(* Schneider Machine Expert - Basic project cb(1), file version 2.6.0.0 *)
(* ProjectInformations: Name=New project *)

HARDWARE
  Cpu 0: TM221CE40R
  EthernetConfiguration: NetworkName=M221, IpAllocationMode=FixedAddress, IpAddress=192.168.0.2, SubnetMask=255.255.255.0
  SerialLineConfiguration: Baud=Baud19200, Parity=ParityEven, DataBits=DataBits8, StopBits=StopBits1, PhysicalMedium=PhysicalMediumRs485, TransmissionMode=TransmissionModeModbusRtu, SlaveId=1, Addressing=SlaveAddressing
  MastTask: UsePeriodScanMode=false, PeriodScan=100
  FastTask: Period=255
  CpuBehavior: StartingMode=StartAsPreviousState, AutoSaveRamOnEeprom=true, WatchdogPeriod=250

SYMBOLS  (address, symbol, comment, settings)
  %M0         "START"
  %M1         "MOVE_TRF"
  %M2         "GRIPPER_C_CLOSE"
  %M3         "MOVE_BACK_TRF"
  %M4         "GRIPPER_ROTATE_CLOSE"
  %M5         "STATUS CB ON"
  %M6         "RELEASE_C_GRIPPER"
  %M7         "POLARITY_ RESULT"
  %M8         "POLARITY_CHECK"
  %M9         "ROTATE_0"
  %M10        "REVERSE_ROTATION"
  %M11        "RESET"
  %M12        "MANUAL"
  %M13        "CB_LF"
  %M14        "CB_RT"
  %M15        "DELAY_CUT_LEFT"
  %M16        "Cut Left"
  %M17        "Cut Right"
  %M19        "Grimp Comp"
  %M20        "R_Grip"
  %M21        "Slide"
  %M22        "LF_CB"
  %M23        "M_Q1"
  %M24        "M_Q2"
  %M25        "M_Q3"
  %M26      MANUAL_GRIP_CLOSE  "M_Q4"
  %M27      SLIDER  "M_Q5"
  %M28        "M_Q6"
  %M29        "Manual Bowl"
  %M30        "EMG_Memory"
  %M31        "Start_Memory"
  %M47        "M_EMG"
  %M49        "POLARITY CHECKED"
  %M50        "NEGATIVE"
  %M51        "POSITIVE"
  %M52        "FIRST RUN"
  %M53        "DONE CUTTING"
  %M54        "NEGATIVE READY"
  %M55        "TRIGGER"
  %M56        "COUNTER OUTPUT"
  %M100       "START GUI"
  %M102       "M_START"
  %MW0        "Count Output"
  %TM0        [Preset=50, Base=TenMilliSeconds]
  %TM1        [Preset=10, Base=TenMilliSeconds]
  %TM2        "Left Cut"  [Preset=10, Base=TenMilliSeconds]
  %I0.0       "EMG"
  %I0.1       "BTN START"
  %I0.2       "LF_CB_FWD"
  %I0.3       "LF_CB_BWD"
  %I0.4       "RT_CB_FWD"
  %I0.5       "RT_CB_BWD"
  %I0.6       "R_CW"
  %I0.7       "R_CCW"
  %I0.8       "GRIP_R_OPEN"
  %I0.9       "GRIP_R_CLOSE"
  %I0.10      "GRIP_C_OPEN"
  %I0.11      "GRIP_C_CLOSE"
  %I0.12      "C_TRF_FWD"
  %I0.13      "TRF_C_BWD"
  %I0.14      "PART_DETECTION"
  %I0.15      "GRIP_C_OPEN"
  %I0.16      "GRIP_C_OPEN"
  %I0.19      "BUTTON POLARITY"
  %Q0.0       "LF_CB"
  %Q0.1       "RT_CB"
  %Q0.2       "R_P"
  %Q0.3       "GRIP_COMP"
  %Q0.4       "GRIP_ROTATE"
  %Q0.5       "TRF_C"
  %Q0.6       "BOWL_FEEDER"

POU New POU
  (* SectionNumber=1 *)

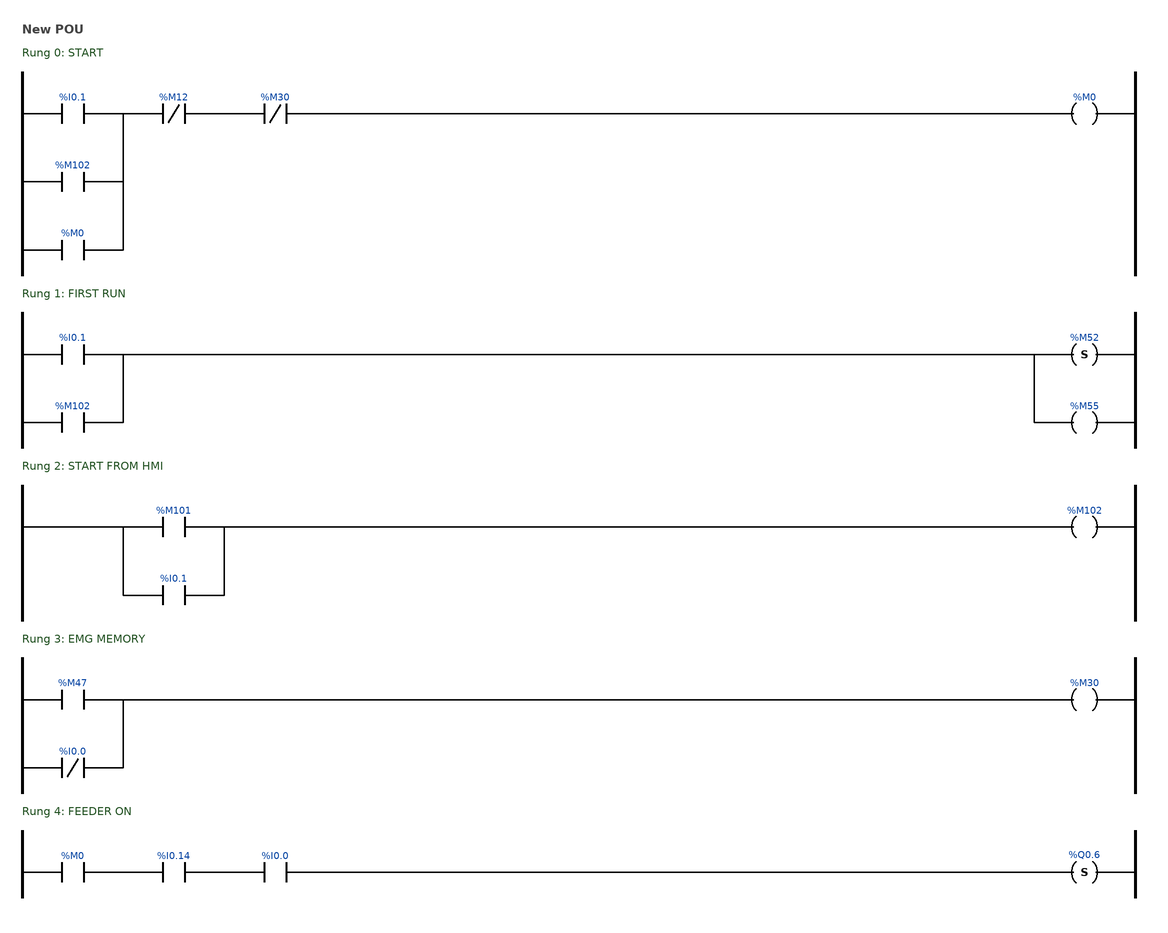

// Rung 0: START
  LD %I0.1
  OR %M102
  OR %M0
  ANDN %M12
  ANDN %M30
  ST %M0
  // as ST:
  //   %M0 := (%I0.1 OR %M102 OR %M0) AND NOT %M12 AND NOT %M30;

// Rung 1: FIRST RUN
  LD %I0.1
  OR %M102
  S %M52
  ST %M55
  // as ST:
  //   IF %I0.1 OR %M102 THEN %M52 := TRUE; END_IF;
  //   %M55 := %I0.1 OR %M102;

// Rung 2: START FROM HMI
  LD 1
  AND( %M101
  OR %I0.1
  )
  ST %M102
  // as ST:
  //   %M102 := %M101 OR %I0.1;

// Rung 3: EMG MEMORY
  LD %M47
  ORN %I0.0
  ST %M30
  // as ST:
  //   %M30 := %M47 OR NOT %I0.0;

// Rung 4: FEEDER ON
  LD %M0
  AND %I0.14
  AND %I0.0
  S %Q0.6
  // as ST:
  //   IF %M0 AND %I0.14 AND %I0.0 THEN %Q0.6 := TRUE; END_IF;

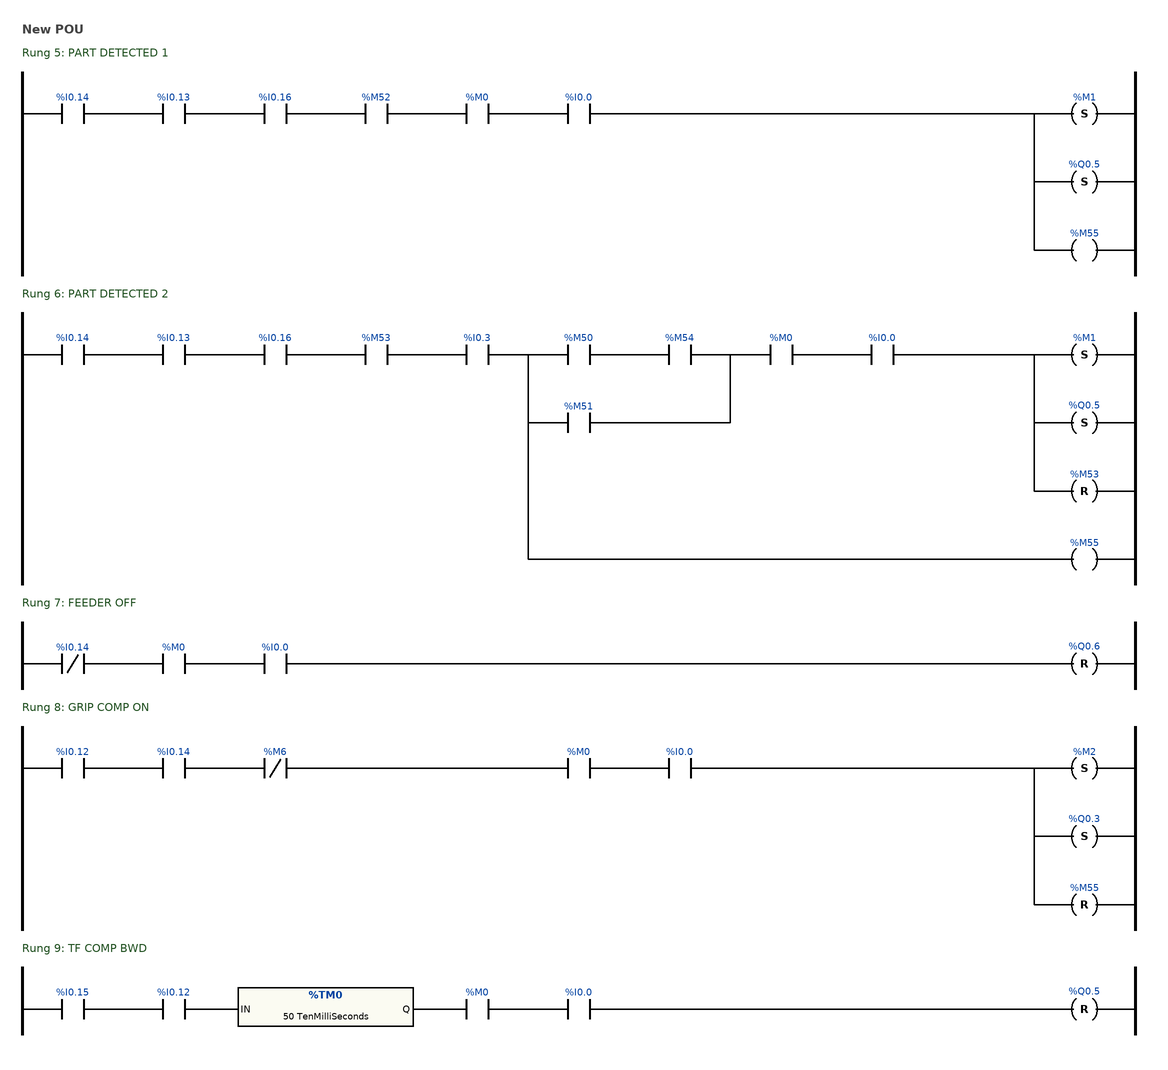

// Rung 5: PART DETECTED 1
  LD %I0.14
  AND %I0.13
  AND %I0.16
  AND %M52
  AND %M0
  AND %I0.0
  S %M1
  S %Q0.5
  ST %M55
  // as ST:
  //   IF %I0.14 AND %I0.13 AND %I0.16 AND %M52 AND %M0 AND %I0.0 THEN %M1 := TRUE; END_IF;
  //   IF %I0.14 AND %I0.13 AND %I0.16 AND %M52 AND %M0 AND %I0.0 THEN %Q0.5 := TRUE; END_IF;
  //   %M55 := %I0.14 AND %I0.13 AND %I0.16 AND %M52 AND %M0 AND %I0.0;

// Rung 6: PART DETECTED 2
  LD %I0.14
  AND %I0.13
  AND %I0.16
  AND %M53
  AND %I0.3
  MPS
  AND( %M50
  AND %M54
  OR %M51
  )
  AND %M0
  AND %I0.0
  S %M1
  S %Q0.5
  R %M53
  MPP
  ST %M55
  // as ST:
  //   IF %I0.14 AND %I0.13 AND %I0.16 AND %M53 AND %I0.3 AND (%M50 AND %M54 OR %M51) AND %M0 AND %I0.0 THEN %M1 := TRUE; END_IF;
  //   IF %I0.14 AND %I0.13 AND %I0.16 AND %M53 AND %I0.3 AND (%M50 AND %M54 OR %M51) AND %M0 AND %I0.0 THEN %Q0.5 := TRUE; END_IF;
  //   _t1 := %I0.14 AND %I0.13 AND %I0.16 AND %M53 AND %I0.3;
  //   IF %I0.14 AND %I0.13 AND %I0.16 AND %M53 AND %I0.3 AND (%M50 AND %M54 OR %M51) AND %M0 AND %I0.0 THEN %M53 := FALSE; END_IF;
  //   %M55 := _t1;

// Rung 7: FEEDER OFF
  LDN %I0.14
  AND %M0
  AND %I0.0
  R %Q0.6
  // as ST:
  //   IF NOT %I0.14 AND %M0 AND %I0.0 THEN %Q0.6 := FALSE; END_IF;

// Rung 8: GRIP COMP ON
  LD %I0.12
  AND %I0.14
  ANDN %M6
  AND %M0
  AND %I0.0
  S %M2
  S %Q0.3
  R %M55
  // as ST:
  //   IF %I0.12 AND %I0.14 AND NOT %M6 AND %M0 AND %I0.0 THEN %M2 := TRUE; END_IF;
  //   IF %I0.12 AND %I0.14 AND NOT %M6 AND %M0 AND %I0.0 THEN %Q0.3 := TRUE; END_IF;
  //   IF %I0.12 AND %I0.14 AND NOT %M6 AND %M0 AND %I0.0 THEN %M55 := FALSE; END_IF;

// Rung 9: TF COMP BWD
  BLK %TM0
  LD %I0.15
  AND %I0.12
  IN
  OUT_BLK
  LD Q
  AND %M0
  AND %I0.0
  R %Q0.5
  END_BLK
  // as ST:
  //   %TM0(IN := %I0.15 AND %I0.12);
  //   IF %TM0.Q AND %M0 AND %I0.0 THEN %Q0.5 := FALSE; END_IF;

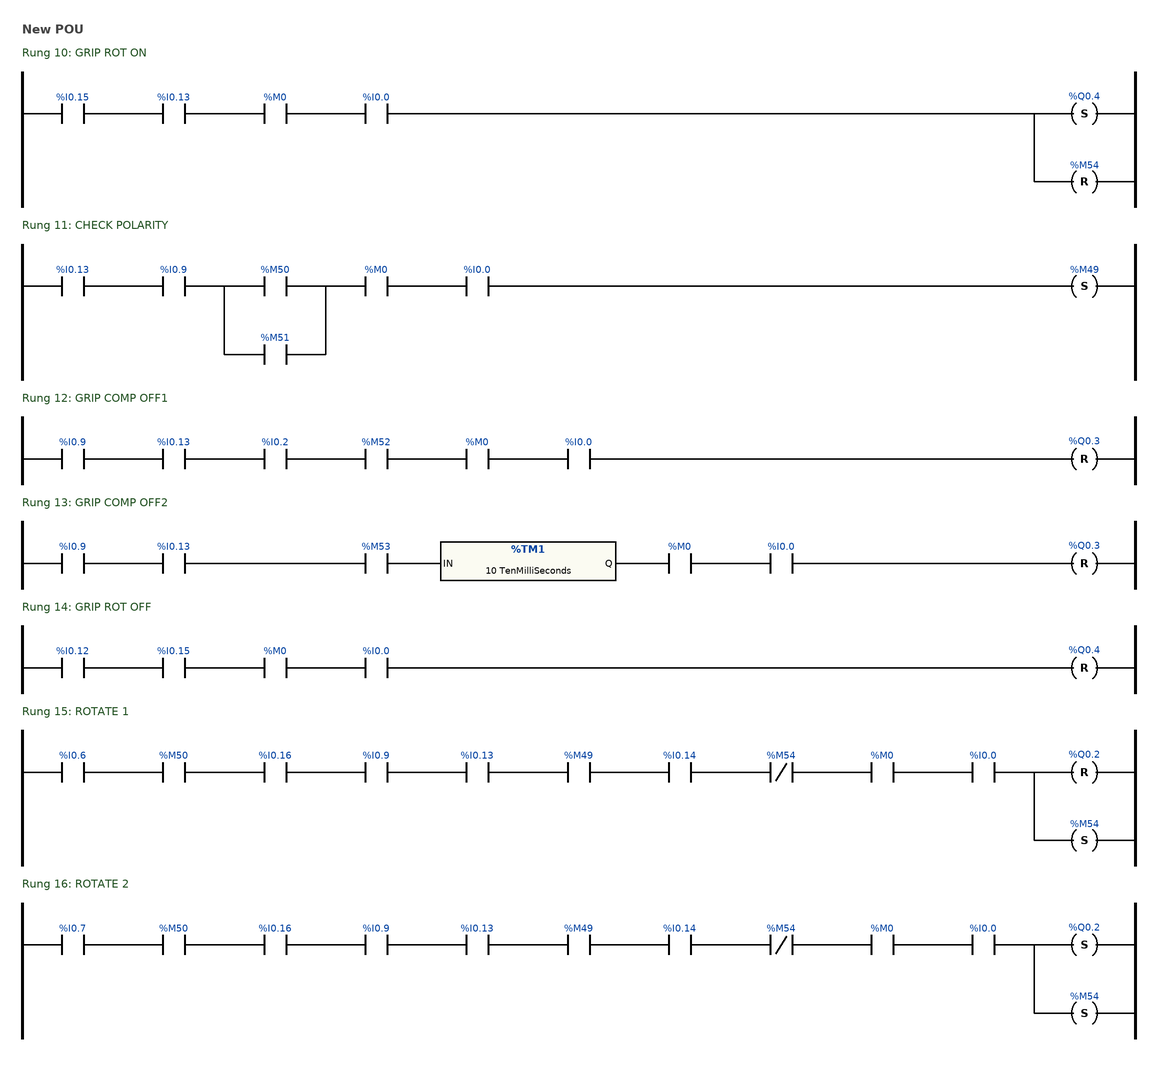

// Rung 10: GRIP ROT ON
  LD %I0.15
  AND %I0.13
  AND %M0
  AND %I0.0
  S %Q0.4
  R %M54
  // as ST:
  //   IF %I0.15 AND %I0.13 AND %M0 AND %I0.0 THEN %Q0.4 := TRUE; END_IF;
  //   IF %I0.15 AND %I0.13 AND %M0 AND %I0.0 THEN %M54 := FALSE; END_IF;

// Rung 11: CHECK POLARITY
  LD %I0.13
  AND %I0.9
  AND( %M50
  OR %M51
  )
  AND %M0
  AND %I0.0
  S %M49
  // as ST:
  //   IF %I0.13 AND %I0.9 AND (%M50 OR %M51) AND %M0 AND %I0.0 THEN %M49 := TRUE; END_IF;

// Rung 12: GRIP COMP OFF1
  LD %I0.9
  AND %I0.13
  AND %I0.2
  AND %M52
  AND %M0
  AND %I0.0
  R %Q0.3
  // as ST:
  //   IF %I0.9 AND %I0.13 AND %I0.2 AND %M52 AND %M0 AND %I0.0 THEN %Q0.3 := FALSE; END_IF;

// Rung 13: GRIP COMP OFF2
  BLK %TM1
  LD %I0.9
  AND %I0.13
  AND %M53
  IN
  OUT_BLK
  LD Q
  AND %M0
  AND %I0.0
  R %Q0.3
  END_BLK
  // as ST:
  //   %TM1(IN := %I0.9 AND %I0.13 AND %M53);
  //   IF %TM1.Q AND %M0 AND %I0.0 THEN %Q0.3 := FALSE; END_IF;

// Rung 14: GRIP ROT OFF
  LD %I0.12
  AND %I0.15
  AND %M0
  AND %I0.0
  R %Q0.4
  // as ST:
  //   IF %I0.12 AND %I0.15 AND %M0 AND %I0.0 THEN %Q0.4 := FALSE; END_IF;

// Rung 15: ROTATE 1
  LD %I0.6
  AND %M50
  AND %I0.16
  AND %I0.9
  AND %I0.13
  AND %M49
  AND %I0.14
  ANDN %M54
  AND %M0
  AND %I0.0
  R %Q0.2
  S %M54
  // as ST:
  //   IF %I0.6 AND %M50 AND %I0.16 AND %I0.9 AND %I0.13 AND %M49 AND %I0.14 AND NOT %M54 AND %M0 AND %I0.0 THEN %Q0.2 := FALSE; END_IF;
  //   IF %I0.6 AND %M50 AND %I0.16 AND %I0.9 AND %I0.13 AND %M49 AND %I0.14 AND NOT %M54 AND %M0 AND %I0.0 THEN %M54 := TRUE; END_IF;

// Rung 16: ROTATE 2
  LD %I0.7
  AND %M50
  AND %I0.16
  AND %I0.9
  AND %I0.13
  AND %M49
  AND %I0.14
  ANDN %M54
  AND %M0
  AND %I0.0
  S %Q0.2
  S %M54
  // as ST:
  //   IF %I0.7 AND %M50 AND %I0.16 AND %I0.9 AND %I0.13 AND %M49 AND %I0.14 AND NOT %M54 AND %M0 AND %I0.0 THEN %Q0.2 := TRUE; END_IF;
  //   IF %I0.7 AND %M50 AND %I0.16 AND %I0.9 AND %I0.13 AND %M49 AND %I0.14 AND NOT %M54 AND %M0 AND %I0.0 THEN %M54 := TRUE; END_IF;

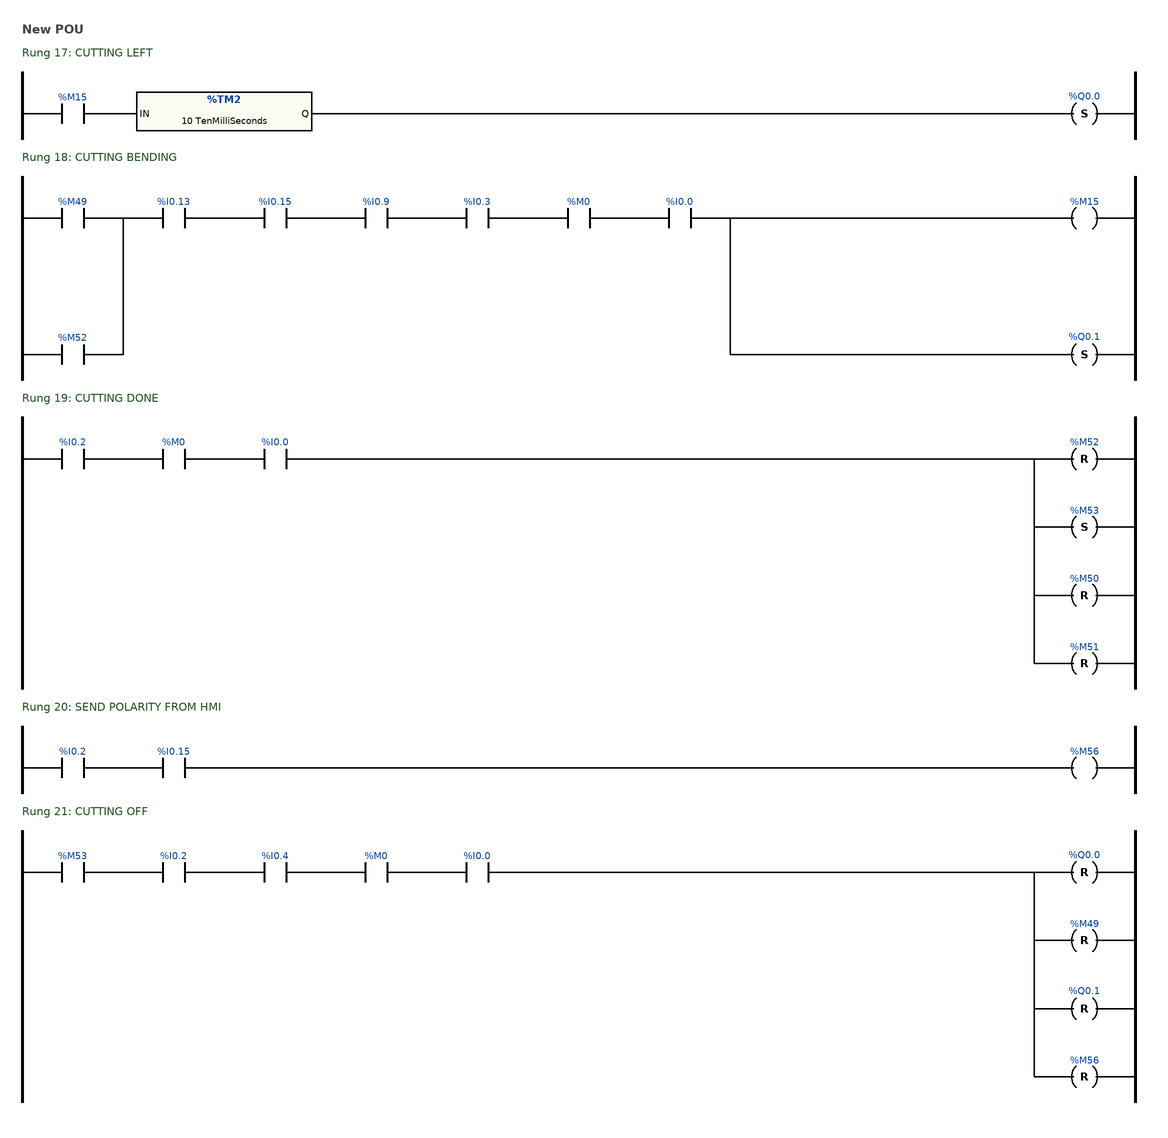

// Rung 17: CUTTING LEFT
  BLK %TM2
  LD %M15
  IN
  OUT_BLK
  LD Q
  S %Q0.0
  END_BLK
  // as ST:
  //   %TM2(IN := %M15);
  //   IF %TM2.Q THEN %Q0.0 := TRUE; END_IF;

// Rung 18: CUTTING BENDING
  LD %M49
  OR %M52
  AND %I0.13
  AND %I0.15
  AND %I0.9
  AND %I0.3
  AND %M0
  AND %I0.0
  ST %M15
  S %Q0.1
  // as ST:
  //   %M15 := (%M49 OR %M52) AND %I0.13 AND %I0.15 AND %I0.9 AND %I0.3 AND %M0 AND %I0.0;
  //   IF (%M49 OR %M52) AND %I0.13 AND %I0.15 AND %I0.9 AND %I0.3 AND %M0 AND %I0.0 THEN %Q0.1 := TRUE; END_IF;

// Rung 19: CUTTING DONE
  LD %I0.2
  AND %M0
  AND %I0.0
  R %M52
  S %M53
  R %M50
  R %M51
  // as ST:
  //   IF %I0.2 AND %M0 AND %I0.0 THEN %M52 := FALSE; END_IF;
  //   IF %I0.2 AND %M0 AND %I0.0 THEN %M53 := TRUE; END_IF;
  //   IF %I0.2 AND %M0 AND %I0.0 THEN %M50 := FALSE; END_IF;
  //   IF %I0.2 AND %M0 AND %I0.0 THEN %M51 := FALSE; END_IF;

// Rung 20: SEND POLARITY FROM HMI
  LD %I0.2
  AND %I0.15
  ST %M56
  // as ST:
  //   %M56 := %I0.2 AND %I0.15;

// Rung 21: CUTTING OFF
  LD %M53
  AND %I0.2
  AND %I0.4
  AND %M0
  AND %I0.0
  R %Q0.0
  R %M49
  R %Q0.1
  R %M56
  // as ST:
  //   IF %M53 AND %I0.2 AND %I0.4 AND %M0 AND %I0.0 THEN %Q0.0 := FALSE; END_IF;
  //   IF %M53 AND %I0.2 AND %I0.4 AND %M0 AND %I0.0 THEN %M49 := FALSE; END_IF;
  //   IF %M53 AND %I0.2 AND %I0.4 AND %M0 AND %I0.0 THEN %Q0.1 := FALSE; END_IF;
  //   IF %M53 AND %I0.2 AND %I0.4 AND %M0 AND %I0.0 THEN %M56 := FALSE; END_IF;

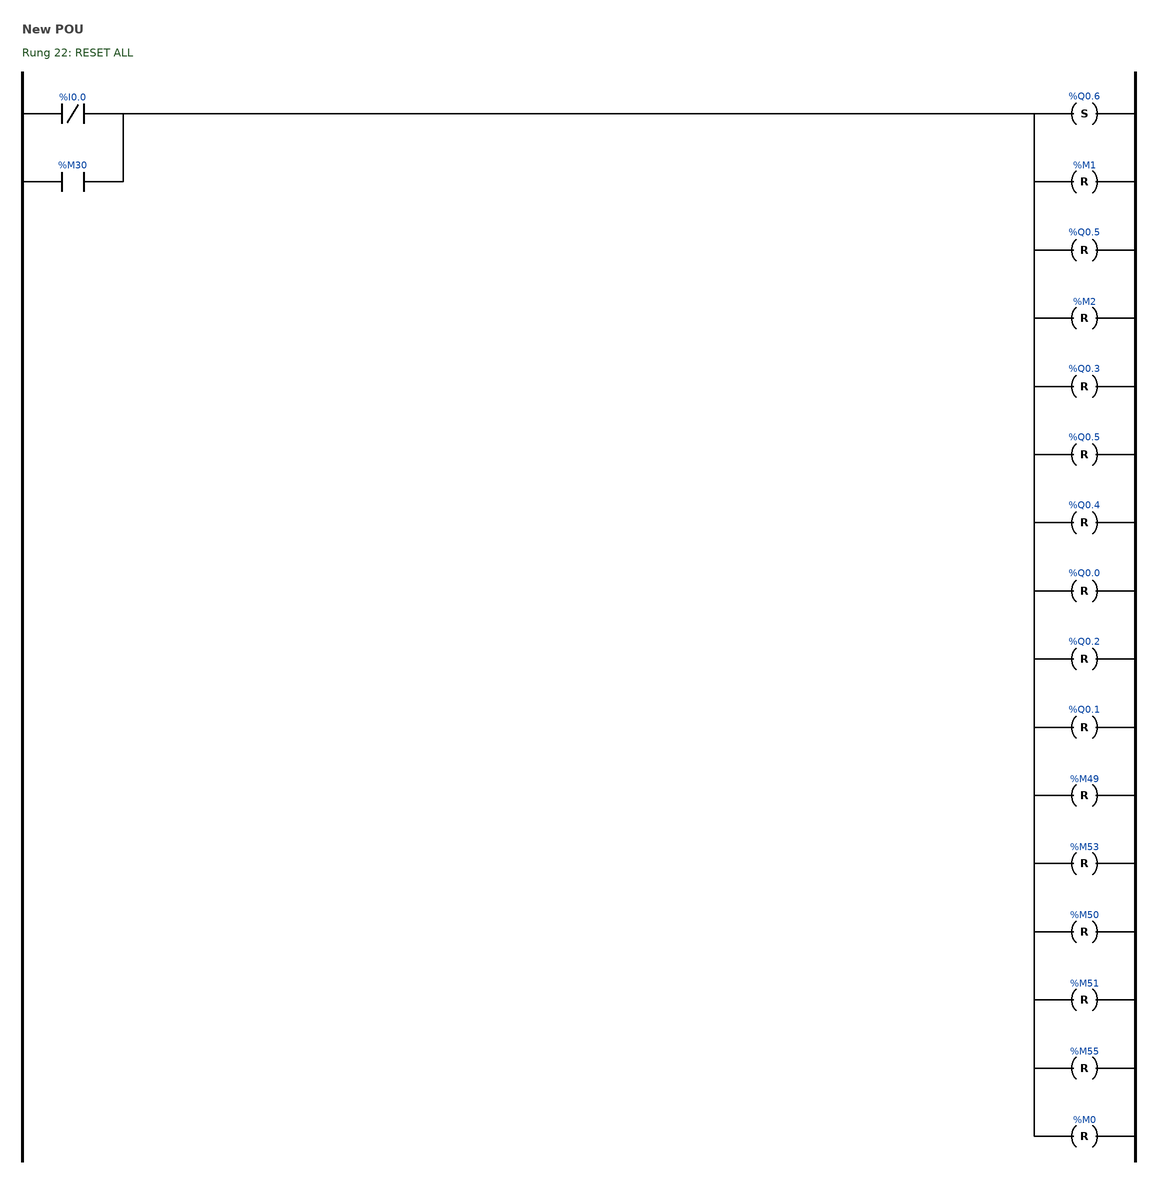

// Rung 22: RESET ALL
  LDN %I0.0
  OR %M30
  S %Q0.6
  R %M1
  R %Q0.5
  R %M2
  R %Q0.3
  R %Q0.5
  R %Q0.4
  R %Q0.0
  R %Q0.2
  R %Q0.1
  R %M49
  R %M53
  R %M50
  R %M51
  R %M55
  R %M0
  // as ST:
  //   IF NOT %I0.0 OR %M30 THEN %Q0.6 := TRUE; END_IF;
  //   IF NOT %I0.0 OR %M30 THEN %M1 := FALSE; END_IF;
  //   IF NOT %I0.0 OR %M30 THEN %Q0.5 := FALSE; END_IF;
  //   IF NOT %I0.0 OR %M30 THEN %M2 := FALSE; END_IF;
  //   IF NOT %I0.0 OR %M30 THEN %Q0.3 := FALSE; END_IF;
  //   IF NOT %I0.0 OR %M30 THEN %Q0.5 := FALSE; END_IF;
  //   IF NOT %I0.0 OR %M30 THEN %Q0.4 := FALSE; END_IF;
  //   IF NOT %I0.0 OR %M30 THEN %Q0.0 := FALSE; END_IF;
  //   IF NOT %I0.0 OR %M30 THEN %Q0.2 := FALSE; END_IF;
  //   IF NOT %I0.0 OR %M30 THEN %Q0.1 := FALSE; END_IF;
  //   IF NOT %I0.0 OR %M30 THEN %M49 := FALSE; END_IF;
  //   IF NOT %I0.0 OR %M30 THEN %M53 := FALSE; END_IF;
  //   IF NOT %I0.0 OR %M30 THEN %M50 := FALSE; END_IF;
  //   IF NOT %I0.0 OR %M30 THEN %M51 := FALSE; END_IF;
  //   IF NOT %I0.0 OR %M30 THEN %M55 := FALSE; END_IF;
  //   IF NOT %I0.0 OR %M30 THEN %M0 := FALSE; END_IF;

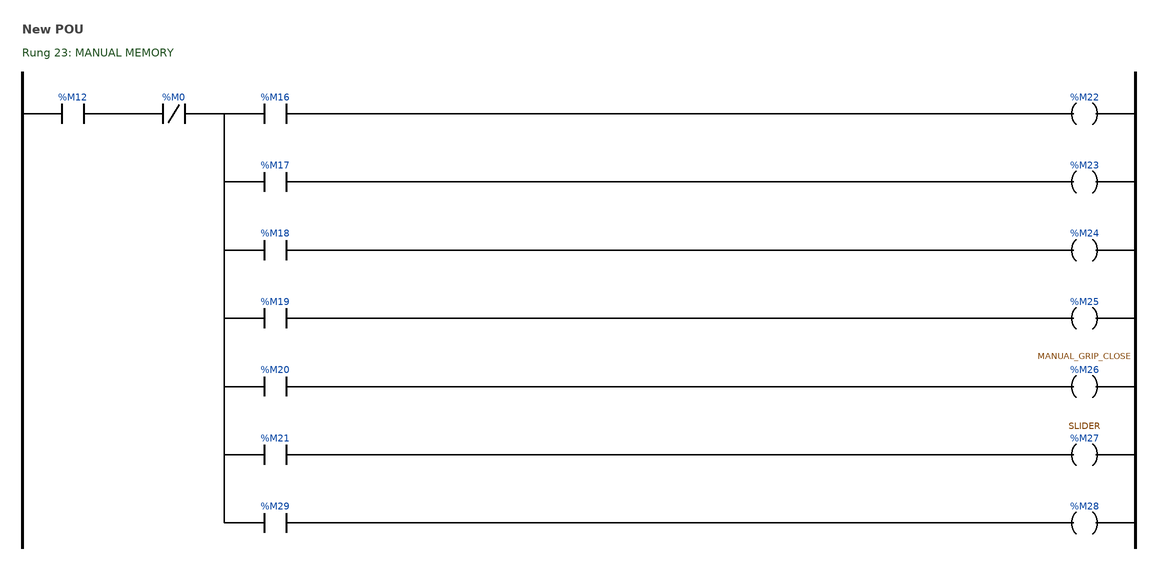

// Rung 23: MANUAL MEMORY
  LD %M12
  ANDN %M0
  MPS
  AND %M16
  ST %M22
  MRD
  AND %M17
  ST %M23
  MRD
  AND %M18
  ST %M24
  MRD
  AND %M19
  ST %M25
  MRD
  AND %M20
  ST %M26                 (* MANUAL_GRIP_CLOSE *)
  MRD
  AND %M21
  ST %M27                 (* SLIDER *)
  MPP
  AND %M29
  ST %M28
  // as ST:
  //   %M22 := %M12 AND NOT %M0 AND %M16;
  //   %M23 := %M12 AND NOT %M0 AND %M17;
  //   %M24 := %M12 AND NOT %M0 AND %M18;
  //   %M25 := %M12 AND NOT %M0 AND %M19;
  //   MANUAL_GRIP_CLOSE := %M12 AND NOT %M0 AND %M20;
  //   SLIDER := %M12 AND NOT %M0 AND %M21;
  //   %M28 := %M12 AND NOT %M0 AND %M29;

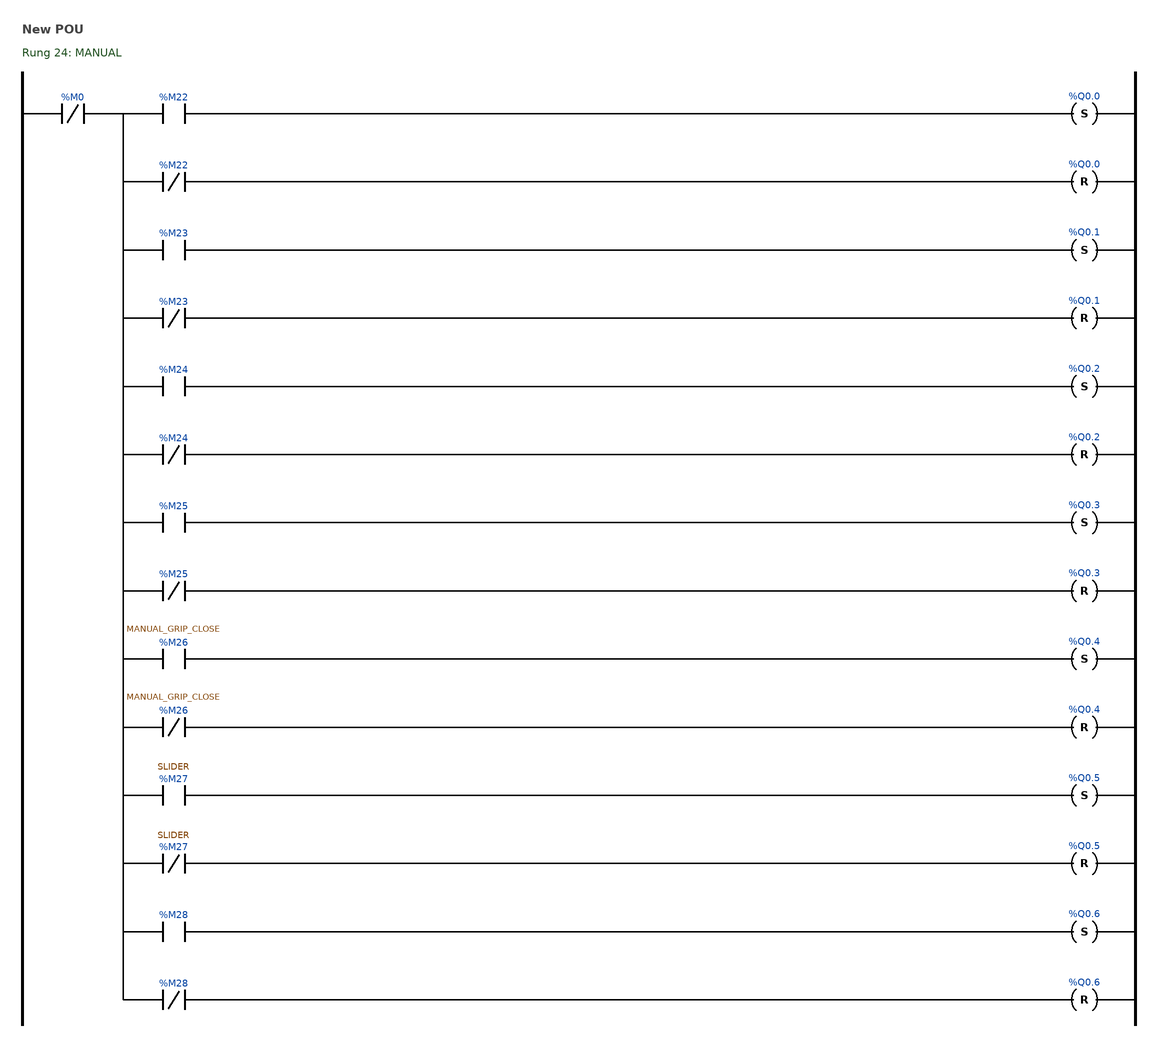

// Rung 24: MANUAL
  LDN %M0
  MPS
  AND %M22
  S %Q0.0
  MRD
  ANDN %M22
  R %Q0.0
  MRD
  AND %M23
  S %Q0.1
  MRD
  ANDN %M23
  R %Q0.1
  MRD
  AND %M24
  S %Q0.2
  MRD
  ANDN %M24
  R %Q0.2
  MRD
  AND %M25
  S %Q0.3
  MRD
  ANDN %M25
  R %Q0.3
  MRD
  AND %M26                (* MANUAL_GRIP_CLOSE *)
  S %Q0.4
  MRD
  ANDN %M26               (* MANUAL_GRIP_CLOSE *)
  R %Q0.4
  MRD
  AND %M27                (* SLIDER *)
  S %Q0.5
  MRD
  ANDN %M27               (* SLIDER *)
  R %Q0.5
  MRD
  AND %M28
  S %Q0.6
  MPP
  ANDN %M28
  R %Q0.6
  // as ST:
  //   IF NOT %M0 AND %M22 THEN %Q0.0 := TRUE; END_IF;
  //   IF NOT %M0 AND NOT %M22 THEN %Q0.0 := FALSE; END_IF;
  //   IF NOT %M0 AND %M23 THEN %Q0.1 := TRUE; END_IF;
  //   IF NOT %M0 AND NOT %M23 THEN %Q0.1 := FALSE; END_IF;
  //   IF NOT %M0 AND %M24 THEN %Q0.2 := TRUE; END_IF;
  //   IF NOT %M0 AND NOT %M24 THEN %Q0.2 := FALSE; END_IF;
  //   IF NOT %M0 AND %M25 THEN %Q0.3 := TRUE; END_IF;
  //   IF NOT %M0 AND NOT %M25 THEN %Q0.3 := FALSE; END_IF;
  //   IF NOT %M0 AND MANUAL_GRIP_CLOSE THEN %Q0.4 := TRUE; END_IF;
  //   IF NOT %M0 AND NOT MANUAL_GRIP_CLOSE THEN %Q0.4 := FALSE; END_IF;
  //   IF NOT %M0 AND SLIDER THEN %Q0.5 := TRUE; END_IF;
  //   IF NOT %M0 AND NOT SLIDER THEN %Q0.5 := FALSE; END_IF;
  //   IF NOT %M0 AND %M28 THEN %Q0.6 := TRUE; END_IF;
  //   IF NOT %M0 AND NOT %M28 THEN %Q0.6 := FALSE; END_IF;

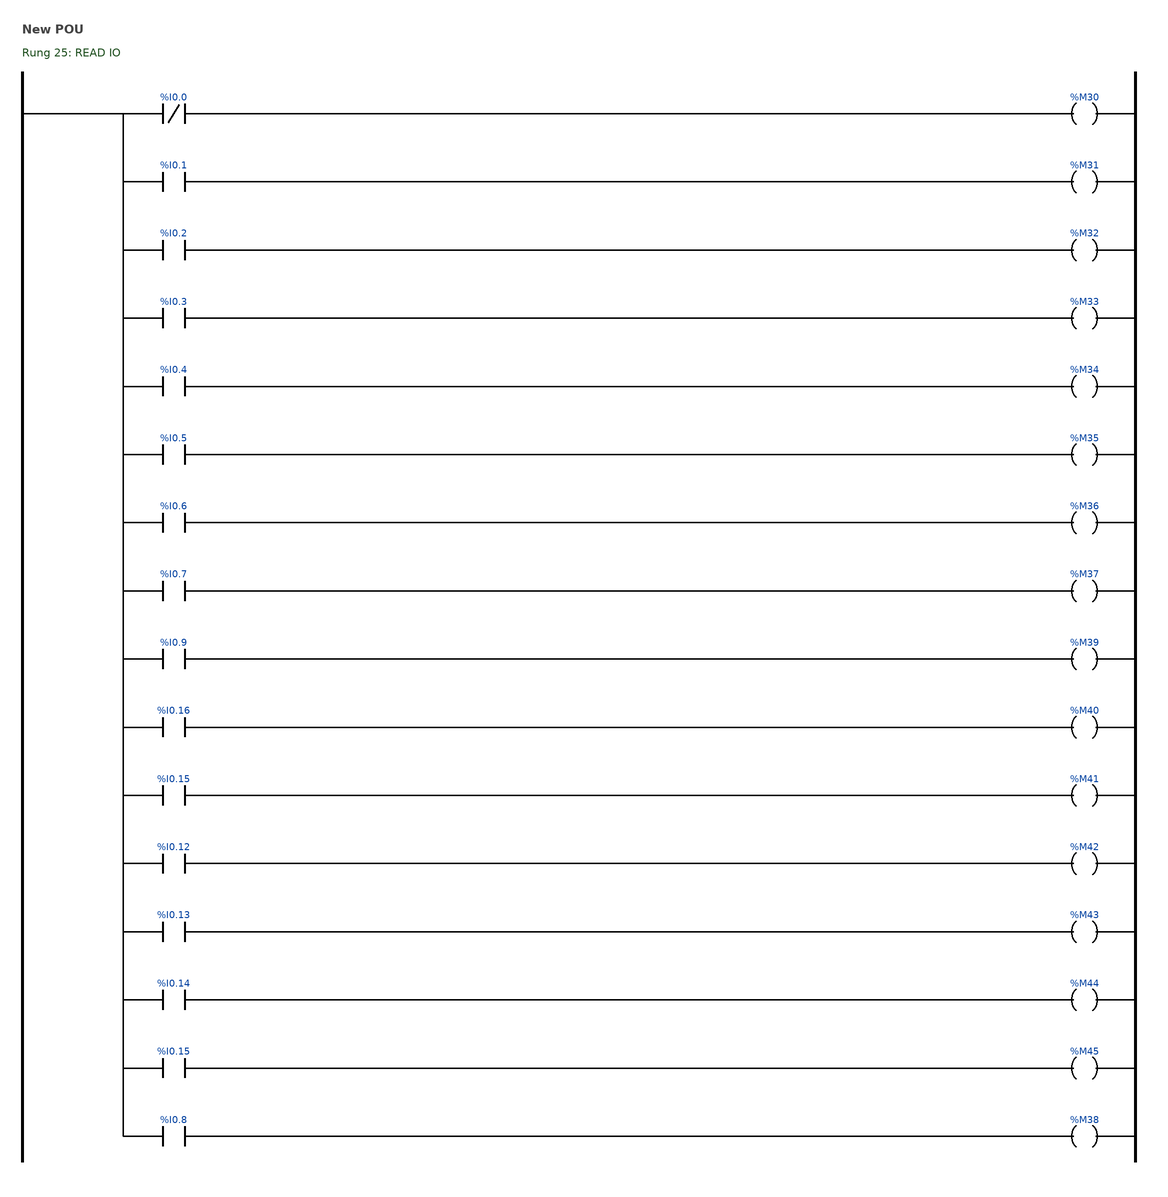

// Rung 25: READ IO
  LD 1
  MPS
  ANDN %I0.0
  ST %M30
  MRD
  AND %I0.1
  ST %M31
  MRD
  AND %I0.2
  ST %M32
  MRD
  AND %I0.3
  ST %M33
  MRD
  AND %I0.4
  ST %M34
  MRD
  AND %I0.5
  ST %M35
  MRD
  AND %I0.6
  ST %M36
  MRD
  AND %I0.7
  ST %M37
  MRD
  AND %I0.9
  ST %M39
  MRD
  AND %I0.16
  ST %M40
  MRD
  AND %I0.15
  ST %M41
  MRD
  AND %I0.12
  ST %M42
  MRD
  AND %I0.13
  ST %M43
  MRD
  AND %I0.14
  ST %M44
  MRD
  AND %I0.15
  ST %M45
  MPP
  AND %I0.8
  ST %M38
  // as ST:
  //   %M30 := NOT %I0.0;
  //   %M31 := %I0.1;
  //   %M32 := %I0.2;
  //   %M33 := %I0.3;
  //   %M34 := %I0.4;
  //   %M35 := %I0.5;
  //   %M36 := %I0.6;
  //   %M37 := %I0.7;
  //   %M39 := %I0.9;
  //   %M40 := %I0.16;
  //   %M41 := %I0.15;
  //   %M42 := %I0.12;
  //   %M43 := %I0.13;
  //   %M44 := %I0.14;
  //   %M45 := %I0.15;
  //   %M38 := %I0.8;
